// TIA Portal V18 export
FUNCTION "PC_connection_main" : Void   // FC8, FBD
{ S7_Optimized_Access := 'TRUE' }
VERSION : 0.1
// stored: AutoNumber true, IsIECCheckEnabled false, SetENOAutomatically false, UDAEnableTagReadback false
   VAR_TEMP
      er_PC_connection : Bool;
   END_VAR
BEGIN

REGION Network 1
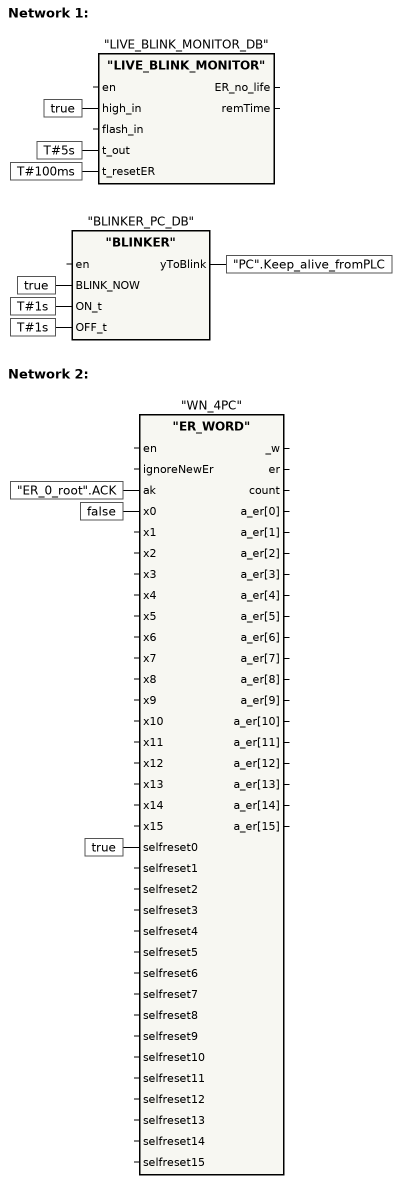
   "LIVE_BLINK_MONITOR_DB"(high_in := true, t_out := T#5s, t_resetER := T#100ms);   // "LIVE_BLINK_MONITOR"
   "BLINKER_PC_DB"(BLINK_NOW := true, ON_t := T#1s, OFF_t := T#1s, yToBlink => "PC".Keep_alive_fromPLC);   // "BLINKER"
END_REGION

REGION Network 2
   "WN_4PC"(ak := "ER_0_root".ACK, x0 := false, selfreset0 := true);   // "ER_WORD"
END_REGION

REGION Network 3
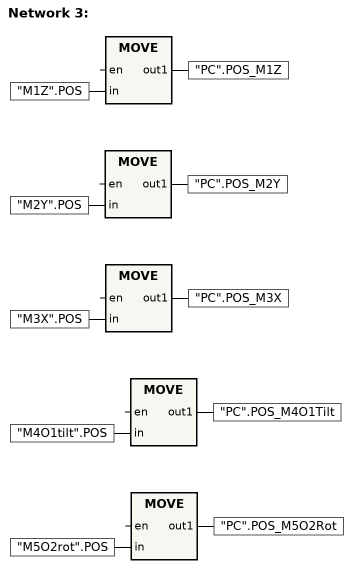
   "PC".POS_M1Z := "M1Z".POS;
   "PC".POS_M2Y := "M2Y".POS;
   "PC".POS_M3X := "M3X".POS;
   "PC".POS_M4O1Tilt := "M4O1tilt".POS;
   "PC".POS_M5O2Rot := "M5O2rot".POS;
END_REGION

REGION Network 4 (SCL)
   %DB69. := %DB69.;
   //%DB69.DBX2.0 := "PC".X_ray_ready_fromPLC;
   //"PC".Image_ready_fromPC := %DB69.DBX4.0;

   IF "PC".PLC_RESET_Image_ready_fromPC THEN
       "PC".Image_ready_fromPC := false;
   END_IF;
END_REGION

REGION Network 6 (SCL)
   (*"PC".POS_M1ZINT := REAL_TO_INT("PC".POS_M1Z);
   "PC".POS_M2YINT := REAL_TO_INT("PC".POS_M2Y);
   "PC".POS_M3XINT := REAL_TO_INT("PC".POS_M3X);
   "PC".POS_M4O1TiltINT := REAL_TO_INT("PC".POS_M4O1TiltINT);
   "PC".POS_M5O2Rot := REAL_TO_INT("PC".POS_M5O2RotINT);*)
END_REGION
END_FUNCTION
